(* Logix 5000 project; controller WWTP_SEC_CLX vendor 1 type 14 code 54 rev 17.2; software revision 17.00 *)
// WWTP Secondary Treatment System

TASK MainTask (continuous, watchdog 500 ms) : MainProgram, SecTank01_Drive, SecTank02_Drive, AerationBlower, SecTank01_RAS_Pump

MODULES
   Local : vendor 1 type 14 code 54 (ICP 0, rev 17.2)
      WWTP_SEC_CLX_Rack00_Slot02_DI : 1756-IA16 (ICP 2, rev 3.2, Input RPI 20 ms)
           Local:2:I.DATA.4   // Secondary Tank #1 In-Auto
           Local:2:I.DATA.7   // Secondary Tank #2 In-Auto
           Local:2:I.DATA.0   // BLR-400 In-Auto
           Local:2:I.DATA.1   // BLR-400 Running
           Local:2:I.DATA.14   // M-401 In-Auto
           Local:2:I.DATA.10   // M-400 Fault
           Local:2:I.DATA.11   // M-400 In-Auto
           Local:2:I.DATA.12   // M-401 Running
           Local:2:I.DATA.13   // M-401 Fault
           Local:2:I.DATA.2   // BLR-400 Fault
           Local:2:I.DATA.9   // M-400 Running
           Local:2:I.DATA.5   // Secondary Tank #1 Torque
           Local:2:I.DATA.8   // Secondary Tank #2 Torque
           Local:2:I.DATA.6   // Secondary Tank #2 Running
           Local:2:I.DATA.3   // Secondary Tank #1 Running
      WWTP_SEC_CLS_Rack00_Slot03_DI : 1756-IA16 (ICP 3, rev 3.2, Input RPI 20 ms)
           Local:3:I.DATA.4   // M-403 Fault
           Local:3:I.DATA.5   // M-403 In-Auto
           Local:3:I.DATA.0   // M-402 Running
           Local:3:I.DATA.3   // M-403 Running
           Local:3:I.DATA.1   // M-402 Fault
           Local:3:I.DATA.2   // M-402 In-Auto
      WWTP_SEC_CLX_Rack00_Slot04_DO : vendor 1 type 7 code 13 (ICP 4, rev 3.2, Output RPI 20 ms)
           Local:4:O.DATA.5   // M-402 Start/Stop
           Local:4:O.DATA.1   // Secondary Tank #2 Start/Stop
           Local:4:O.DATA.2   // BLR-400 Start/Stop
           Local:4:O.DATA.3   // M-400 Start/Stop
           Local:4:O.DATA.4   // M-401 Start/Stop
           Local:4:O.DATA.0   // Secondary Tank #1 Start/Stop
           Local:4:O.DATA.6   // M-403 Start/Stop
      WWTP_SEC_CLX_Rack00_Slot05_AI : 1756-IF16 (ICP 5, rev 1.5, Input RPI 100 ms)
           Local:5:I.CH1DATA   // Secondary Tank #2 RAS Control 0 - 3 MGD
           Local:5:I.CH0DATA   // Secondary Tank #1 RAS Control 0 - 3 MGD
      WWTP_SEC_CLX_Rack00_Slot01_ENBT : 1756-ENBT (Ethernet 10.16.3.230, ICP 1, rev 4.2)
         WWTP_RAS_P401 : vendor 1 type 123 code 104 (Ethernet 10.16.3.233, rev 6.4, Output RPI 20 ms)
END_MODULES

TYPE STRING_16 :
STRUCT
   LEN : DINT;
   DATA : SINT[16];
END_STRUCT
END_TYPE

TYPE STRING_20 :
STRUCT
   LEN : DINT;
   DATA : SINT[20];
END_STRUCT
END_TYPE

TYPE STRING_40 :
STRUCT
   LEN : DINT;
   DATA : SINT[40];
END_STRUCT
END_TYPE

TYPE STRING_8 :
STRUCT
   LEN : DINT;
   DATA : SINT[8];
END_STRUCT
END_TYPE

ADD_ON_INSTRUCTION P_AIn   (* revision 0.31, ExecutePrescan, ExecuteEnableInFalse *)
// Analog Input
// Revision note:
// Fixed handling of +/- Inf (1.$) and +/- NaN (1.#QNAN) on Val_InpPV, Val, and filter.
// Help:
// This Instruction monitors an Analog Input from a flow, level, pressure,
// temperature, or any other analog sensor, and provides:
// *  Scaling, from Input (Raw) to PV (Engineering) Units
// *  High-High, High, Low and Low-Low Alarms with configurable delay times and deadbands
// *  Monitoring of input uncertain/bad variable/communication status and out-of-range conditions with alarm
// *  Setting of a simulated input signal for process simulation
// Modes of operation: Operator, Program, Maintenance
// *  Program and Operator Settings for Alarm Thresholds
// *  Maintenance Commands to allow manual override of the input signal (Substitute PV)
VAR_INPUT
   Inp_PV : REAL; {visible}   // Input Signal (process variable) from Sensor
   Inp_PVBad : BOOL;   // 1=PV or I/O Comms Status Bad, 0=OK
   Inp_PVUncertain : BOOL;   // 1=PV Value Not Reliable, 0=OK
   Inp_Sim : BOOL;   // 1=Use simulated PV (Set_SimPV); 0=Use Input (Inp_PV)
   Inp_Reset : BOOL;   // 1=Reset all Alarms requiring reset
   Cfg_NoSubstPV : BOOL;   // 1=Disallow selection of Substitute PV
   Cfg_SetTrack : BOOL := 1;   // 1=PSets track OSets in Oper, OSets track PSets in Prog, 0=no tracking
   Cfg_PCmdClear : BOOL := 1;   // 1=Clear Program Commands on receipt 0=Leave Set
   Cfg_HasHiHiAlm : BOOL;   // 1=High-High Alarm exists and will be checked
   Cfg_HasHiAlm : BOOL;   // 1=High Alarm exists and will be checked
   Cfg_HasLoAlm : BOOL;   // 1=Low Alarm exists and will be checked
   Cfg_HasLoLoAlm : BOOL;   // 1=Low-Low Alarm exists and will be checked
   Cfg_HasFailAlm : BOOL;   // 1=Analog Input Failure Alarm exists and will be checked
   Cfg_HiHiResetReqd : BOOL;   // 1=Reset required to clear High-High Alarm
   Cfg_HiResetReqd : BOOL;   // 1=Reset required to clear High Alarm
   Cfg_LoResetReqd : BOOL;   // 1=Reset required to clear Low Alarm
   Cfg_LoLoResetReqd : BOOL;   // 1=Reset required to clear Low-Low Alarm
   Cfg_FailResetReqd : BOOL;   // 1=Reset required to clear Analog InputFailure Alarm
   Cfg_HiHiAckReqd : BOOL := 1;   // 1=Acknowledge required for High-High Alarm
   Cfg_HiAckReqd : BOOL := 1;   // 1=Acknowledge required for High Alarm
   Cfg_LoAckReqd : BOOL := 1;   // 1=Acknlowledge required for Low Alarm
   Cfg_LoLoAckReqd : BOOL := 1;   // 1=Acknowledge required for Low-Low Alarm
   Cfg_FailAckReqd : BOOL := 1;   // 1=Acknowledge required for Analog Input Failure Alarm
   Cfg_HiHiSeverity : SINT := 3;   // High-High Alarm Severity 1=info, 2=warn, 3=excep, 4=fault
   Cfg_HiSeverity : SINT := 2;   // High Alarm Severity 1=info, 2=warn, 3=excep, 4=fault
   Cfg_LoSeverity : SINT := 2;   // Low Alarm Severity 1=info, 2=warn, 3=excep, 4=fault
   Cfg_LoLoSeverity : SINT := 3;   // Low-Low Alarm Severity 1=info, 2=warn, 3=excep, 4=fault
   Cfg_FailSeverity : SINT := 4;   // Failure Alarm Severity 1=info, 2=warn, 3=excep, 4=fault
   Cfg_InpRawMin : REAL;   // Input (unscaled) Minimum for Scaling
   Cfg_InpRawMax : REAL := 100.0;   // Input (unscaled) Maximum for Scaling
   Cfg_PVEUMin : REAL;   // PV (Output) Minimum for Scaling to EU
   Cfg_PVEUMax : REAL := 100.0;   // PV (Output) Maximum for Scaling to EU
   Cfg_FiltTC : REAL;   // PV Filter Time Constant (sec), 0.0 = unfiltered
   Cfg_HiHiDB : REAL := 1.0;   // High-High Alarm Deadband (EU)
   Cfg_HiHiMinDuration : DINT;   // Minimum time above High-High Limit to raise Alarm (sec)
   Cfg_HiDB : REAL := 1.0;   // High Alarm Deadband (EU)
   Cfg_HiMinDuration : DINT;   // Minimum time above High Limit to raise Alarm (sec)
   Cfg_LoDB : REAL := 1.0;   // Low Alarm Deadband (EU)
   Cfg_LoMinDuration : DINT;   // Minimum time below Low Limit to raise Alarm (sec)
   Cfg_LoLoDB : REAL := 1.0;   // Low-Low Alarm Deadband (EU)
   Cfg_LoLoMinDuration : DINT;   // Minimum time below Low-Low Limit to raise Alarm (sec)
   Cfg_FailHiLim : REAL := 1.5e+38;   // Out-of-Range (fail) High Limit (EU)
   Cfg_FailLoLim : REAL := -1.5e+38;   // Out-of-Range (fail) Low Limit (EU)
   Cfg_FailDB : REAL;   // Out-of-Range (fail) High/Low Deadband (EU)
   Cfg_FailMinDuration : DINT;   // Minimum time Bad or Out of Range to raise Fail Alarm (sec)
   PSet_Owner : DINT;   // Program Owner Request ID (non-zero) or Release (zero)
   PSet_HiHiLim : REAL := 1.5e+38;   // Program-Entered High-High Alarm Threshold (EU)
   PSet_HiLim : REAL := 1.5e+38;   // Program-Entered High Alarm Threshold (EU)
   PSet_LoLim : REAL := -1.5e+38;   // Program-Entered Low Alarm Threshold (EU)
   PSet_LoLoLim : REAL := -1.5e+38;   // Program-Entered Low-Low Alarm Threshold (EU)
   MSet_SubstPV : REAL;   // Maintenance-Entered Substitute PV (EU)
   OSet_HiHiLim : REAL := 1.5e+38;   // Operator-Entered High-High Alarm Threshold (EU)
   OSet_HiLim : REAL := 1.5e+38;   // Operator-Entered High Alarm Threshold (EU)
   OSet_LoLim : REAL := -1.5e+38;   // Operator-Entered Low Alarm Threshold (EU)
   OSet_LoLoLim : REAL := -1.5e+38;   // Operator-Entered Low-Low Alarm Threshold (EU)
   Set_SimPV : REAL;   // PV used in Simulation (Inp_Sim=1) (EU)
   PCmd_Acq : BOOL;   // Program Command to Acquire ownership (Oper to Prog)
   PCmd_Rel : BOOL;   // Program Command to Release ownership (Prog to Oper)
   PCmd_Lock : BOOL;   // Program Command to Lock Mode in Prog
   PCmd_Unlock : BOOL;   // Program Command to Unlock Mode
   PCmd_Reset : BOOL;   // Program Command to Reset all Alarms requiring Reset
   PCmd_HiHiAck : BOOL;   // Program Command to Acknowledge High-High Alarm
   PCmd_HiHiInhibit : BOOL;   // Program Command to Inhibit High-High Alarm
   PCmd_HiHiUninhibit : BOOL;   // Program Command to UninhibitHigh-High Alarm
   PCmd_HiAck : BOOL;   // Program Command to Acknowledge High Alarm
   PCmd_HiInhibit : BOOL;   // Program Command to Inhibit High Alarm
   PCmd_HiUninhibit : BOOL;   // Program Command to Uninhibit High Alarm
   PCmd_LoAck : BOOL;   // Program Command to Acknowledge Low Alarm
   PCmd_LoInhibit : BOOL;   // Program Command to Inhibit Low Alarm
   PCmd_LoUninhibit : BOOL;   // Program Command to Uninhibit Low Alarm
   PCmd_LoLoAck : BOOL;   // Program Command to Acknowledge Low-Low Alarm
   PCmd_LoLoInhibit : BOOL;   // Program Command to Inhibit Low-Low Alarm
   PCmd_LoLoUninhibit : BOOL;   // Program Command to Uninhibit Low-Low Alarm
   PCmd_FailAck : BOOL;   // Program Command to Acknowldege Analog Input Failure Alarm
   PCmd_FailInhibit : BOOL;   // Program Command to Inhibit Analog Input Failure Alarm
   PCmd_FailUninhibit : BOOL;   // Program Command to Uninhibit Analog Input Failure Alarm
   MCmd_SubstPV : BOOL;   // Maintenance Command to use Substitute PV (override input)
   MCmd_InpPV : BOOL;   // Maintenance Command to use Input PV (normal)
   OCmd_Reset : BOOL;   // Operator Command to Reset all Alarms requiring Reset
END_VAR
VAR_OUTPUT
   Val : REAL; {visible}   // Analog Value (after Substitute PV, if used)
   Val_InpPV : REAL; {visible}   // Analog Input Value (actual, before Substitute PV selection)
   Val_PVEUMin : REAL;   // Minimum of scaled range = MIN (Cfg_PVEUMin, Cfg_PVEUMax)
   Val_PVEUMax : REAL := 100.0;   // Maximum of scaled range = MAX (Cfg_PVEUMin, Cfg_PVEUMax)
   Val_Owner : DINT;   // Current Object Owner ID (0=not owned)
   Val_Notify : SINT;   // Current Alarm Level and Acknowledgement (enumeration)
   Val_HiHiLim : REAL := 1.5e+38; {visible}   // Current High-High Alarm Threshold
   Val_HiLim : REAL := 1.5e+38; {visible}   // Current High Alarm Threshold
   Val_LoLim : REAL := -1.5e+38; {visible}   // Current Low Alarm Threshold
   Val_LoLoLim : REAL := -1.5e+38; {visible}   // Current Low-Low Alarm Threshold
   Sts_SubstPV : BOOL;   // 1=Using Substitute PV (Input being overridden)
   Sts_InpPV : BOOL := 1;   // 1=Using Input PV (normal)
   Sts_PVBad : BOOL;   // 1=PV Bad quality or Out of Range
   Sts_PVUncertain : BOOL;   // 1=PV Value is Uncertain (quality)
   Sts_Err : BOOL; {visible}   // 1=Error in Config, see detail Err_ bits for reason
   Err_Raw : BOOL;   // 1=Error in Config: Raw Input Scaling Min = Max
   Err_EU : BOOL;   // 1=Error in Config: Scaled EU Min = Max
   Err_Filt : BOOL;   // 1=Error in Config: PV filter params (RateTime, TC)
   Err_DB : BOOL;   // 1=Error in Config: an Alarm Deadband is < 0.0
   Err_Alarm : BOOL;   // 1=Error in Config: Invalid Alarm Min Duration or Severity
   Sts_Maint : BOOL;   // 1=Mode is Maintenance (supersedes Prog, Oper)
   Sts_Prog : BOOL;   // 1=Mode is Program
   Sts_Oper : BOOL := 1;   // 1=Mode is Operator
   Sts_ProgOperLock : BOOL;   // 1=Program or Operator has requested Mode Lock
   Sts_HiHi : BOOL;   // 1=Analog Input is above High-High limit
   Alm_HiHi : BOOL;   // 1=Analog Input is in High-High Alarm
   Ack_HiHi : BOOL;   // 1=High-High Alarm has been acknowledged
   Sts_HiHiDisabled : BOOL;   // 1=High-High Alarm is Disabled (not saved or sent)
   Sts_HiHiInhibited : BOOL;   // 1=High-High Alarm is Inhibited by logic
   Sts_HiHiSuppressed : BOOL;   // 1=High-High Alarm has been suppressed (logged only)
   Sts_Hi : BOOL;   // 1=Analog Input is above High limit
   Alm_Hi : BOOL;   // 1=Analog Input is in High Alarm
   Ack_Hi : BOOL;   // 1=High Alarm has been acknowledged
   Sts_HiDisabled : BOOL;   // 1=High Alarm is Disabled (not saved or sent)
   Sts_HiInhibited : BOOL;   // 1=High Alarm is Inhibited by logic
   Sts_HiSuppressed : BOOL;   // 1=High Alarm has been suppressed (logged only)
   Sts_Lo : BOOL;   // 1=Analog Input is below Low limit
   Alm_Lo : BOOL;   // 1=Analog Input is in Low Alarm
   Ack_Lo : BOOL;   // 1=Low Alarm has been acknowledged
   Sts_LoDisabled : BOOL;   // 1=Low Alarm is Disabled (not saved or sent)
   Sts_LoInhibited : BOOL;   // 1=Low Alarm is Inhibited by logic
   Sts_LoSuppressed : BOOL;   // 1=Low Alarm has been suppressed (logged only)
   Sts_LoLo : BOOL;   // 1=Analog Input is below Low-Low limit
   Alm_LoLo : BOOL;   // 1=Analog Input is in Low-Low Alarm
   Ack_LoLo : BOOL;   // 1=Low-Low Alarm has been acknowledged
   Sts_LoLoDisabled : BOOL;   // 1=Low-Low Alarm is Disabled (not saved or sent)
   Sts_LoLoInhibited : BOOL;   // 1=Low-Low Alarm is Inhibited by logic
   Sts_LoLoSuppressed : BOOL;   // 1=Low-Low Alarm has been suppressed (logged only)
   Sts_Fail : BOOL;   // 1=Analog Input is Out of Range or PV Bad
   Alm_Fail : BOOL;   // 1=Analog Input Failure Alarm (Bad or Out of Range)
   Ack_Fail : BOOL;   // 1=Analog Input Failure Alarm has been acknowledged
   Sts_FailDisabled : BOOL;   // 1=Analog input Failure Alarm is Disabled (not saved or sent)
   Sts_FailInhibited : BOOL;   // 1=Analog Input Failure Alarm is inhibited by logic
   Sts_FailSuppressed : BOOL;   // 1=Analog Input Failure Alarm has been suppressed (logged only)
   Rdy_SubstPV : BOOL;   // 1=Ready for MCmd_SubstPV
   Rdy_InpPV : BOOL;   // 1=Ready for MCmd_InpPV
   Rdy_Reset : BOOL;   // 1=At least one Alarm requires Reset
END_VAR
VAR
   LoLo : P_Alarm := (Inp := 1, Cfg_AckReqd := 1, Cfg_Severity := 3, Ack := 1, Rdy_Disable := 1);   // Low-Low Alarm
   Lo : P_Alarm := (Inp := 1, Cfg_AckReqd := 1, Cfg_Severity := 3, Ack := 1, Rdy_Disable := 1);   // Low Alarm
   Hi : P_Alarm := (Inp := 1, Cfg_AckReqd := 1, Cfg_Severity := 2, Ack := 1, Rdy_Disable := 1);   // High Alarm
   HiHi : P_Alarm := (Inp := 1, Cfg_AckReqd := 1, Cfg_Severity := 3, Ack := 1, Rdy_Disable := 1);   // High-High Alarm
   Mode : P_Mode := (Cfg_PCmdClear := 1, Cfg_OvrdOverLock := 1, Sts_Oper := 1, Rdy_Rel := 1, Rdy_AcqLock := 1);   // Analog Input Mode Selection
   Cfg_EU : STRING_8 := '%';   // Engineering Units for display on HMI
   Cfg_Tag : STRING_20 := 'P_AIn';   // Tagname for display on HMI
   Cfg_Label : STRING_20 := 'Analog Input';   // Label for graphic symbol displayed on HMI
   Cfg_Desc : STRING_40 := 'Analog Input';   // Description for display on HMI
   Fail : P_Alarm := (Inp := 1, Cfg_AckReqd := 1, Cfg_Severity := 3, Ack := 1, Rdy_Disable := 1);   // Analog Input Failure Alarm (bad quality or out of range)
   Wrk_Notify : SINT;   // Buffer for building Val_Notify
   Wrk_SubstPV : BOOL;   // Internal flag: Using Substitute PV
   Wrk_UnfiltPV : REAL;   // Unfiltered PV, input to 1st order filter
   Wrk_Alpha : REAL;   // Filter multiplier = (1 / (1+TC/dT) )
   Wrk_ScanT : TIMER := (PRE := 2147483647);   // Scan Timer (milliseconds, always runs)
   Wrk_ScanTime : REAL;   // Time since this instance was last scanned
   Wrk_FiltPV : REAL;   // Filtered PV
   Wrk_InpDINT : DINT;   // Input REAL bit pattern as a DINT (check for Inf/NaN)
   Wrk_InpInfNaN : BOOL;   // Input is Infinite or Not a Number
   Wrk_ValidONS : BOOL;   // Selected PV goes from Infinite or Not a Number to VALID
   Wrk_SelPVDINT : DINT;   // Selected PV check for Infinite or Non A Number
   Wrk_SelPVInfNaN : BOOL;   // Selected PV (Input or Substitute) is Infinite or NaN
END_VAR

ROUTINE EnableInFalse   (* ladder *)
// Off-Scan: no Val update or alarm checking.  PV Bad Quality ("stale") is asserted.
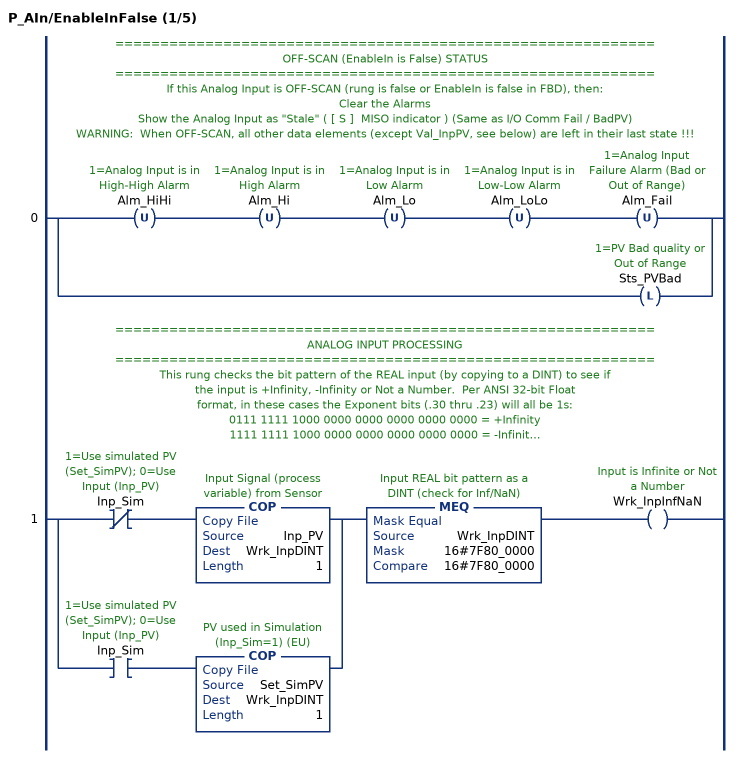
   // ============================================================
   // OFF-SCAN (EnableIn is False) STATUS
   // ============================================================
   // If this Analog Input is OFF-SCAN (rung is false or EnableIn is false in FBD), then:
   // Clear the Alarms
   // Show the Analog Input as "Stale" ( [ S ]  MISO indicator ) (Same as I/O Comm Fail / BadPV)
   // WARNING:  When OFF-SCAN, all other data elements (except Val_InpPV, see below) are left in their last state !!!
   0: [OTU(Alm_HiHi) OTU(Alm_Hi) OTU(Alm_Lo) OTU(Alm_LoLo) OTU(Alm_Fail) ,OTL(Sts_PVBad) ];
   // ============================================================
   // ANALOG INPUT PROCESSING
   // ============================================================
   // This rung checks the bit pattern of the REAL input (by copying to a DINT) to see if
   // the input is +Infinity, -Infinity or Not a Number.  Per ANSI 32-bit Float
   // format, in these cases the Exponent bits (.30 thru .23) will all be 1s:
   // 0111 1111 1000 0000 0000 0000 0000 0000 = +Infinity
   // 1111 1111 1000 0000 0000 0000 0000 0000 = -Infinity
   // x111 1111 1xxx xxxx xxxx xxxx xxxx xxxx = Not a Number
   1: [XIO(Inp_Sim) COP(Inp_PV,Wrk_InpDINT,1) ,XIC(Inp_Sim) COP(Set_SimPV,Wrk_InpDINT,1) ]MEQ(Wrk_InpDINT,16#7F80_0000,16#7F80_0000)OTE(Wrk_InpInfNaN);
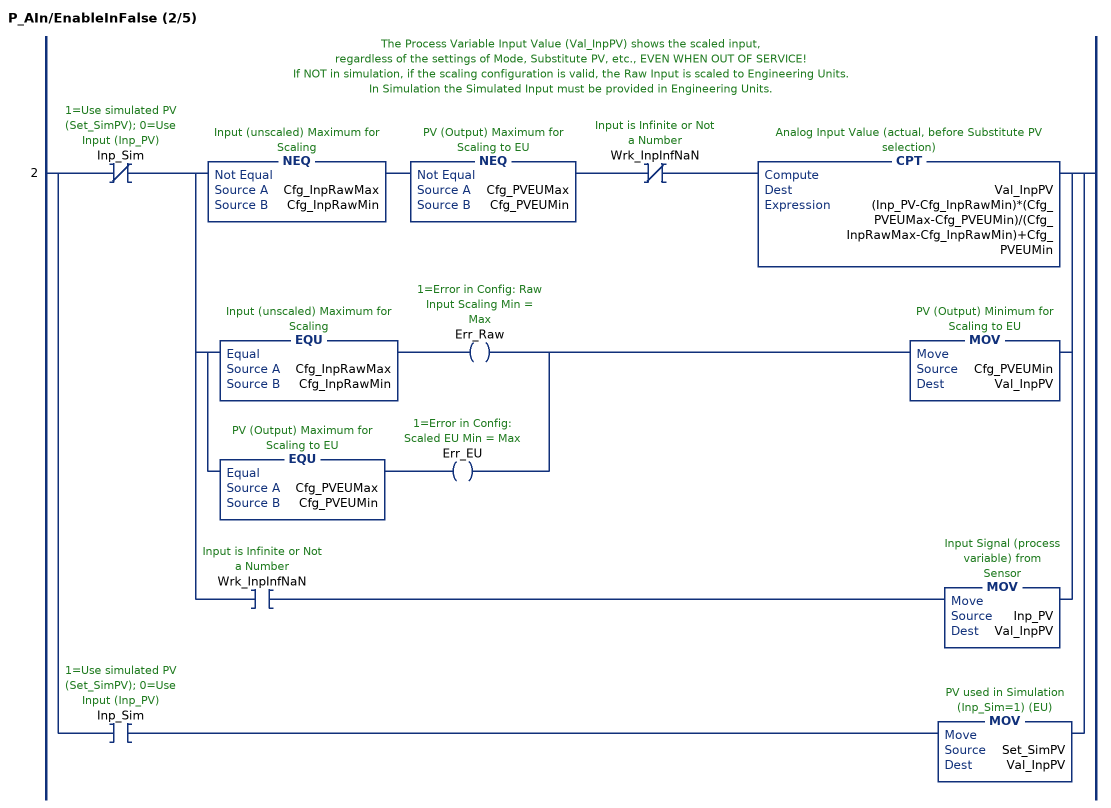
   // The Process Variable Input Value (Val_InpPV) shows the scaled input,
   // regardless of the settings of Mode, Substitute PV, etc., EVEN WHEN OUT OF SERVICE!
   // If NOT in simulation, if the scaling configuration is valid, the Raw Input is scaled to Engineering Units.
   // In Simulation the Simulated Input must be provided in Engineering Units.
   2: [XIO(Inp_Sim) [NEQ(Cfg_InpRawMax,Cfg_InpRawMin) NEQ(Cfg_PVEUMax,Cfg_PVEUMin) XIO(Wrk_InpInfNaN) CPT(Val_InpPV,(Inp_PV-Cfg_InpRawMin)*(Cfg_PVEUMax-Cfg_PVEUMin)/(Cfg_InpRawMax-Cfg_InpRawMin)+Cfg_PVEUMin) ,[EQU(Cfg_InpRawMax,Cfg_InpRawMin) OTE(Err_Raw) ,EQU(Cfg_PVEUMax,Cfg_PVEUMin) OTE(Err_EU) ] MOV(Cfg_PVEUMin,Val_InpPV) ,XIC(Wrk_InpInfNaN) MOV(Inp_PV,Val_InpPV) ] ,XIC(Inp_Sim) MOV(Set_SimPV,Val_InpPV) ];
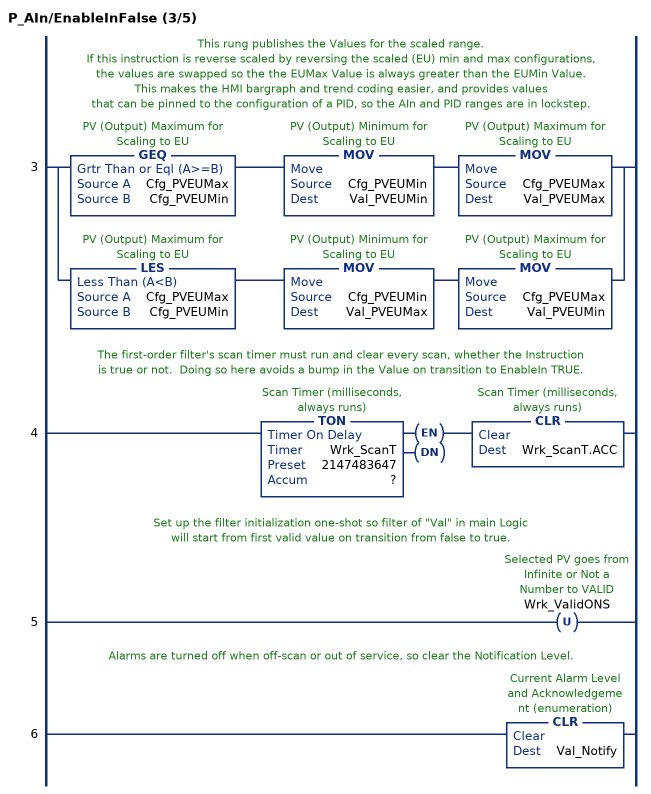
   // This rung publishes the Values for the scaled range.
   // If this instruction is reverse scaled by reversing the scaled (EU) min and max configurations,
   // the values are swapped so the the EUMax Value is always greater than the EUMin Value.
   // This makes the HMI bargraph and trend coding easier, and provides values
   // that can be pinned to the configuration of a PID, so the AIn and PID ranges are in lockstep.
   3: [GEQ(Cfg_PVEUMax,Cfg_PVEUMin) MOV(Cfg_PVEUMin,Val_PVEUMin) MOV(Cfg_PVEUMax,Val_PVEUMax) ,LES(Cfg_PVEUMax,Cfg_PVEUMin) MOV(Cfg_PVEUMin,Val_PVEUMax) MOV(Cfg_PVEUMax,Val_PVEUMin) ];
   // The first-order filter's scan timer must run and clear every scan, whether the Instruction
   // is true or not.  Doing so here avoids a bump in the Value on transition to EnableIn TRUE.
   4: TON(Wrk_ScanT,?,?)CLR(Wrk_ScanT.ACC);
   // Set up the filter initialization one-shot so filter of "Val" in main Logic
   // will start from first valid value on transition from false to true.
   5: OTU(Wrk_ValidONS);
   // Alarms are turned off when off-scan or out of service, so clear the Notification Level.
   6: CLR(Val_Notify);
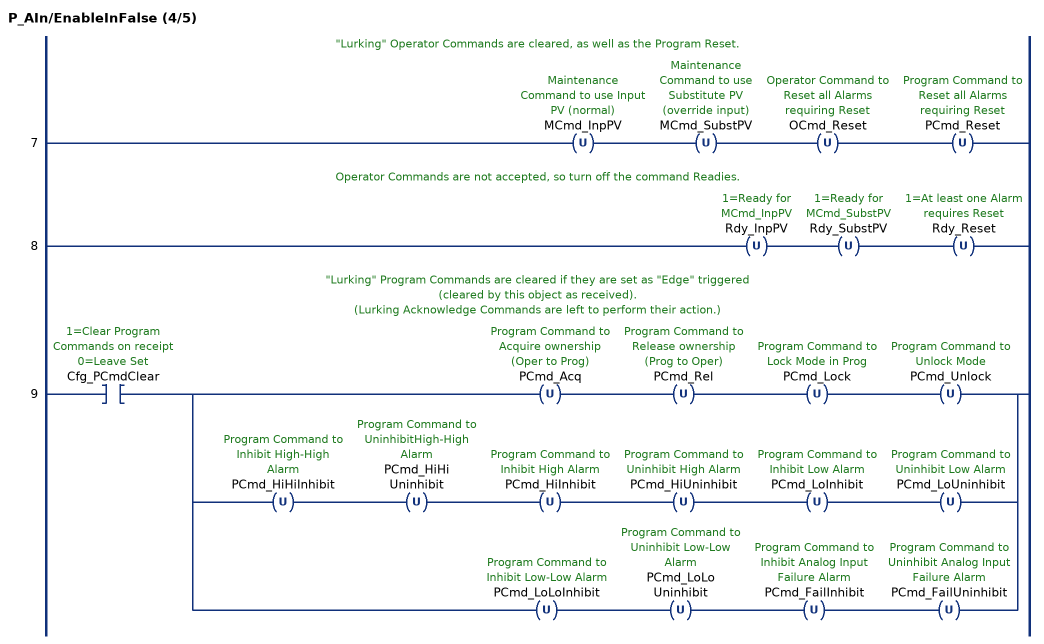
   // "Lurking" Operator Commands are cleared, as well as the Program Reset.
   7: OTU(MCmd_InpPV)OTU(MCmd_SubstPV)OTU(OCmd_Reset)OTU(PCmd_Reset);
   // Operator Commands are not accepted, so turn off the command Readies.
   8: OTU(Rdy_InpPV)OTU(Rdy_SubstPV)OTU(Rdy_Reset);
   // "Lurking" Program Commands are cleared if they are set as "Edge" triggered
   // (cleared by this object as received).
   // (Lurking Acknowledge Commands are left to perform their action.)
   9: XIC(Cfg_PCmdClear)[OTU(PCmd_Acq) OTU(PCmd_Rel) OTU(PCmd_Lock) OTU(PCmd_Unlock) ,OTU(PCmd_HiHiInhibit) OTU(PCmd_HiHiUninhibit) OTU(PCmd_HiInhibit) OTU(PCmd_HiUninhibit) OTU(PCmd_LoInhibit) OTU(PCmd_LoUninhibit) ,OTU(PCmd_LoLoInhibit) OTU(PCmd_LoLoUninhibit) OTU(PCmd_FailInhibit) OTU(PCmd_FailUninhibit) ];
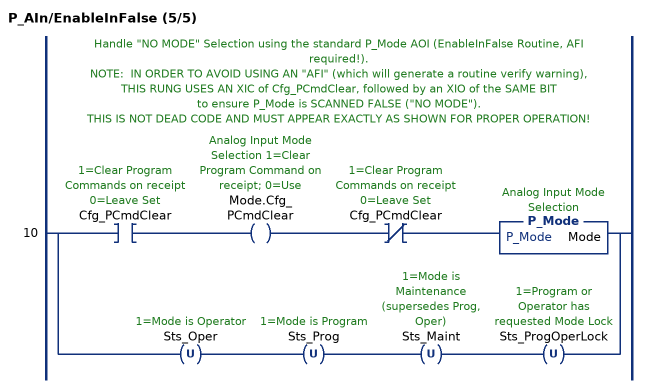
   // Handle "NO MODE" Selection using the standard P_Mode AOI (EnableInFalse Routine, AFI required!).
   // NOTE:  IN ORDER TO AVOID USING AN "AFI" (which will generate a routine verify warning),
   // THIS RUNG USES AN XIC of Cfg_PCmdClear, followed by an XIO of the SAME BIT
   // to ensure P_Mode is SCANNED FALSE ("NO MODE").
   // THIS IS NOT DEAD CODE AND MUST APPEAR EXACTLY AS SHOWN FOR PROPER OPERATION!
   10: [XIC(Cfg_PCmdClear) OTE(Mode.Cfg_PCmdClear) XIO(Cfg_PCmdClear) P_Mode(Mode) ,OTU(Sts_Oper) OTU(Sts_Prog) OTU(Sts_Maint) OTU(Sts_ProgOperLock) ];
END_ROUTINE

ROUTINE Logic   (* ladder *)
// Normal Scan - PV is scaled and alarms are generated
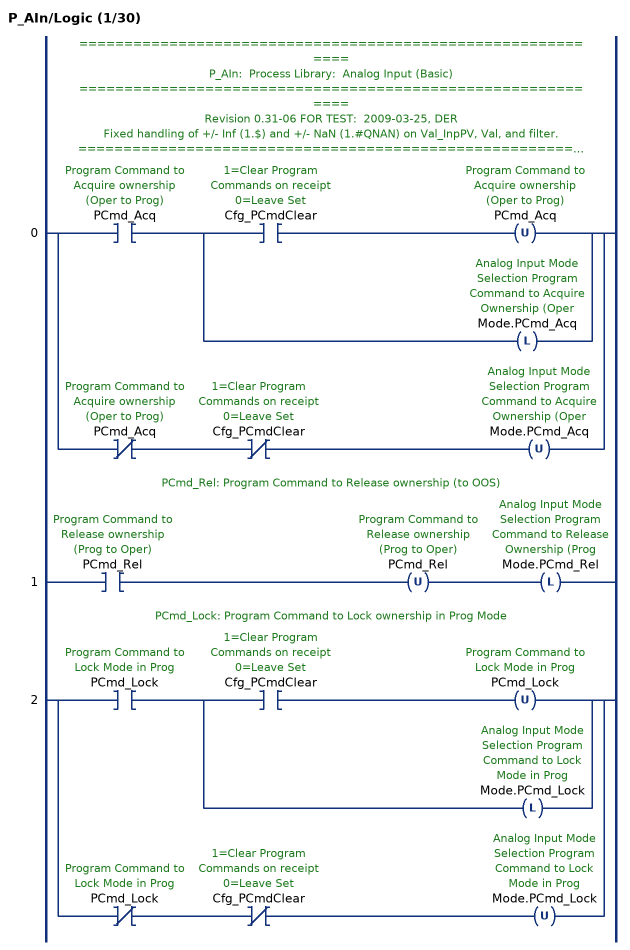
   // ============================================================
   // P_AIn:  Process Library:  Analog Input (Basic)
   // ============================================================
   // Revision 0.31-06 FOR TEST:  2009-03-25, DER
   // Fixed handling of +/- Inf (1.$) and +/- NaN (1.#QNAN) on Val_InpPV, Val, and filter.
   // ============================================================
   // This Instruction monitors an Analog Input from a flow, level, pressure,
   // temperature, or any other analog sensor, and provides:
   // *  Scaling, from Input (Raw) to PV (Engineering) Units
   // *  High-High, High, Low and Low-Low Alarms with configurable delay times and deadbands
   // *  Monitoring of input bad/uncertain variable/communication status and out-of-range conditions with alarm
   // *  Setting of a simulated input signal for process simulation
   // Modes of operation: Operator, Program, Maintenance
   // *  Program and Operator Settings for Alarm Thresholds
   // *  Maintenance Commands to allow manual override of the input signal (Substitute PV)
   // ============================================================
   // POWERUP / INVALID STATE HANDLING
   // ============================================================
   // See Prescan routine for powerup code required for this object.
   // ============================================================
   // MODE PROCESSING
   // ============================================================
   // These rungs handle received Mode Inputs and Commands:
   // NOTE:  Operator Commands for Mode, Alarm are sent directly to the contained P_Mode and P_Alarm AOIs.
   // PCmd_Acq: Program Command to Acquire ownership
   0: [XIC(PCmd_Acq) [XIC(Cfg_PCmdClear) OTU(PCmd_Acq) ,OTL(Mode.PCmd_Acq) ] ,XIO(PCmd_Acq) XIO(Cfg_PCmdClear) OTU(Mode.PCmd_Acq) ];
   // PCmd_Rel: Program Command to Release ownership (to OOS)
   1: XIC(PCmd_Rel)OTU(PCmd_Rel)OTL(Mode.PCmd_Rel);
   // PCmd_Lock: Program Command to Lock ownership in Prog Mode
   2: [XIC(PCmd_Lock) [XIC(Cfg_PCmdClear) OTU(PCmd_Lock) ,OTL(Mode.PCmd_Lock) ] ,XIO(PCmd_Lock) XIO(Cfg_PCmdClear) OTU(Mode.PCmd_Lock) ];
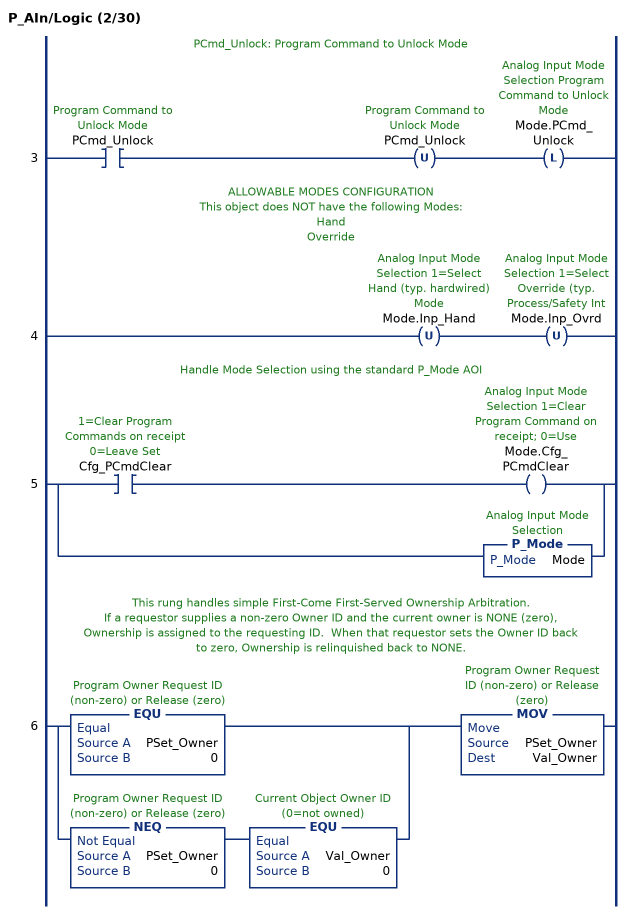
   // PCmd_Unlock: Program Command to Unlock Mode
   3: XIC(PCmd_Unlock)OTU(PCmd_Unlock)OTL(Mode.PCmd_Unlock);
   // ALLOWABLE MODES CONFIGURATION
   // This object does NOT have the following Modes:
   // Hand
   // Override
   4: OTU(Mode.Inp_Hand)OTU(Mode.Inp_Ovrd);
   // Handle Mode Selection using the standard P_Mode AOI
   5: [XIC(Cfg_PCmdClear) OTE(Mode.Cfg_PCmdClear) ,P_Mode(Mode) ];
   // This rung handles simple First-Come First-Served Ownership Arbitration.
   // If a requestor supplies a non-zero Owner ID and the current owner is NONE (zero),
   // Ownership is assigned to the requesting ID.  When that requestor sets the Owner ID back
   // to zero, Ownership is relinquished back to NONE.
   6: [EQU(PSet_Owner,0) ,NEQ(PSet_Owner,0) EQU(Val_Owner,0) ]MOV(PSet_Owner,Val_Owner);
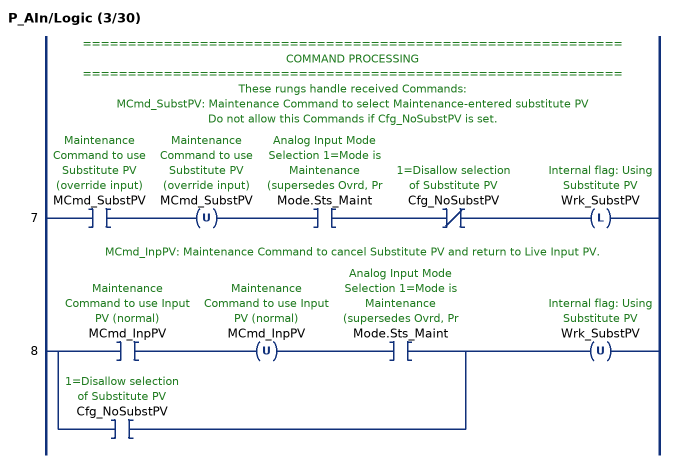
   // ============================================================
   // COMMAND PROCESSING
   // ============================================================
   // These rungs handle received Commands:
   // MCmd_SubstPV: Maintenance Command to select Maintenance-entered substitute PV
   // Do not allow this Commands if Cfg_NoSubstPV is set.
   7: XIC(MCmd_SubstPV)OTU(MCmd_SubstPV)XIC(Mode.Sts_Maint)XIO(Cfg_NoSubstPV)OTL(Wrk_SubstPV);
   // MCmd_InpPV: Maintenance Command to cancel Substitute PV and return to Live Input PV.
   8: [XIC(MCmd_InpPV) OTU(MCmd_InpPV) XIC(Mode.Sts_Maint) ,XIC(Cfg_NoSubstPV) ]OTU(Wrk_SubstPV);
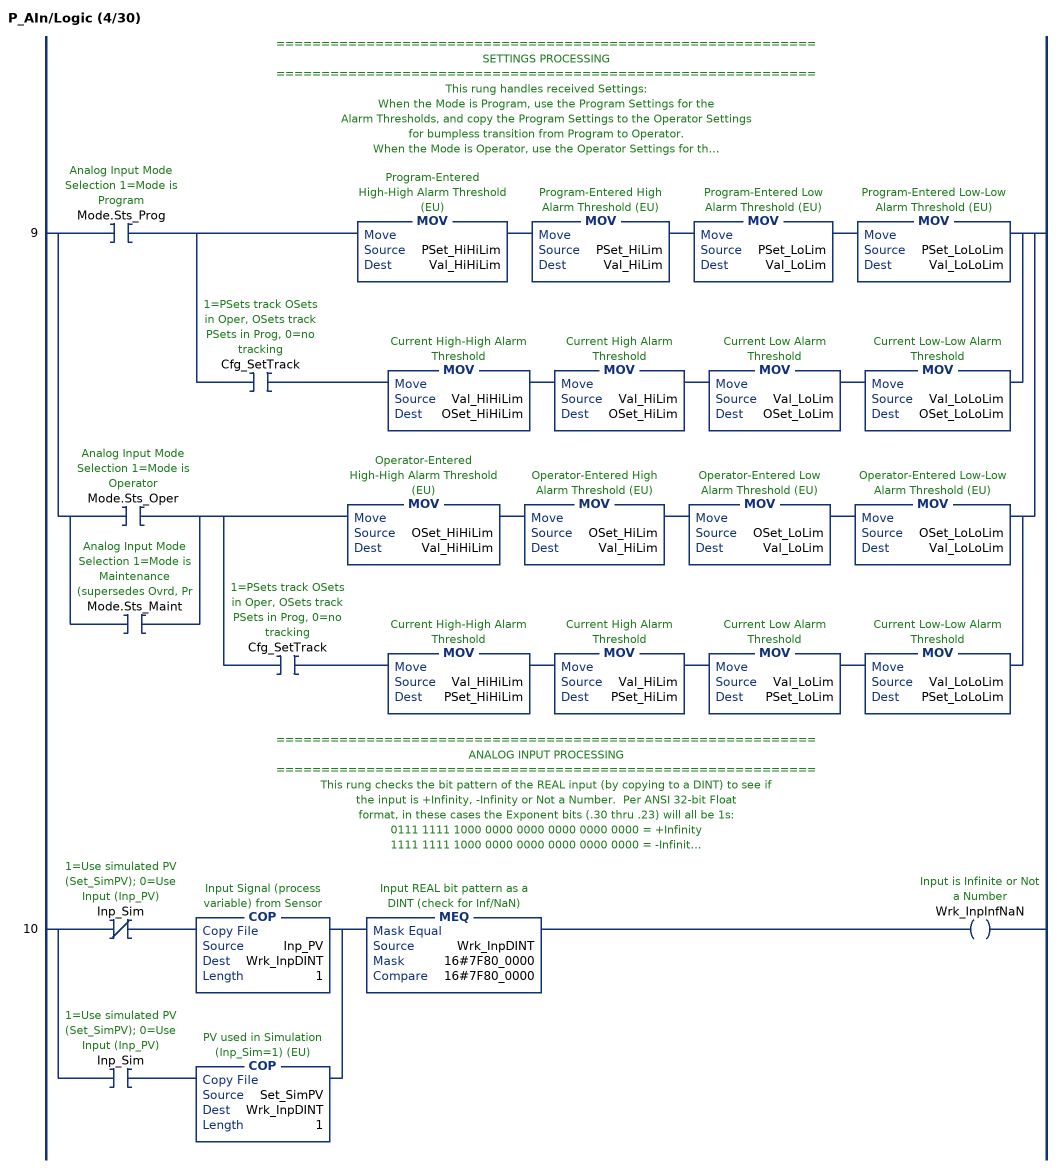
   // ============================================================
   // SETTINGS PROCESSING
   // ============================================================
   // This rung handles received Settings:
   // When the Mode is Program, use the Program Settings for the
   // Alarm Thresholds, and copy the Program Settings to the Operator Settings
   // for bumpless transition from Program to Operator.
   // When the Mode is Operator, use the Operator Settings for the
   // Alarm Thresholds, and copy the Operator Settings to the Program Settings
   // for bumpless transition from Operator to Program.
   9: [XIC(Mode.Sts_Prog) [MOV(PSet_HiHiLim,Val_HiHiLim) MOV(PSet_HiLim,Val_HiLim) MOV(PSet_LoLim,Val_LoLim) MOV(PSet_LoLoLim,Val_LoLoLim) ,XIC(Cfg_SetTrack) MOV(Val_HiHiLim,OSet_HiHiLim) MOV(Val_HiLim,OSet_HiLim) MOV(Val_LoLim,OSet_LoLim) MOV(Val_LoLoLim,OSet_LoLoLim) ] ,[XIC(Mode.Sts_Oper) ,XIC(Mode.Sts_Maint) ] [MOV(OSet_HiHiLim,Val_HiHiLim) MOV(OSet_HiLim,Val_HiLim) MOV(OSet_LoLim,Val_LoLim) MOV(OSet_LoLoLim,Val_LoLoLim) ,XIC(Cfg_SetTrack) MOV(Val_HiHiLim,PSet_HiHiLim) MOV(Val_HiLim,PSet_HiLim) MOV(Val_LoLim,PSet_LoLim) MOV(Val_LoLoLim,PSet_LoLoLim) ] ];
   // ============================================================
   // ANALOG INPUT PROCESSING
   // ============================================================
   // This rung checks the bit pattern of the REAL input (by copying to a DINT) to see if
   // the input is +Infinity, -Infinity or Not a Number.  Per ANSI 32-bit Float
   // format, in these cases the Exponent bits (.30 thru .23) will all be 1s:
   // 0111 1111 1000 0000 0000 0000 0000 0000 = +Infinity
   // 1111 1111 1000 0000 0000 0000 0000 0000 = -Infinity
   // x111 1111 1xxx xxxx xxxx xxxx xxxx xxxx = Not a Number
   10: [XIO(Inp_Sim) COP(Inp_PV,Wrk_InpDINT,1) ,XIC(Inp_Sim) COP(Set_SimPV,Wrk_InpDINT,1) ]MEQ(Wrk_InpDINT,16#7F80_0000,16#7F80_0000)OTE(Wrk_InpInfNaN);
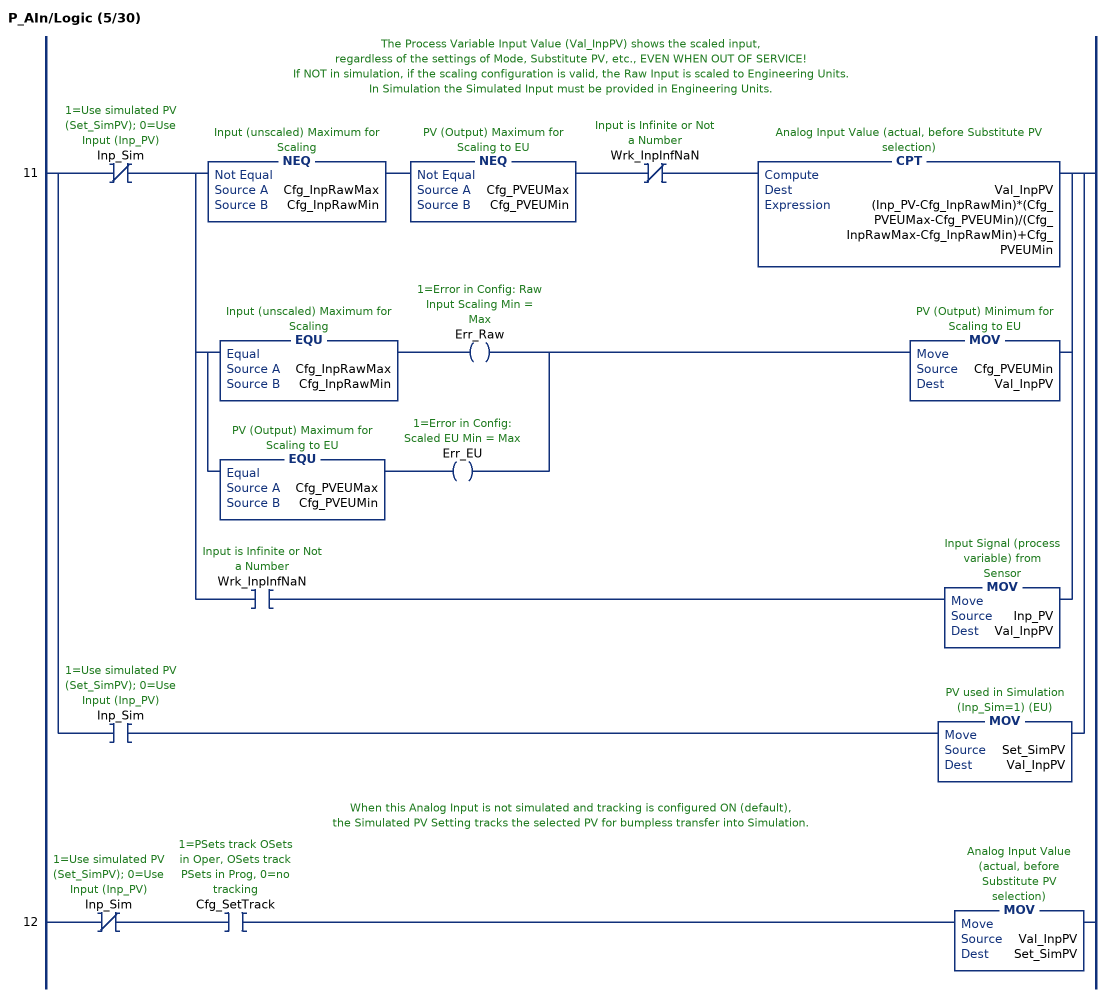
   // The Process Variable Input Value (Val_InpPV) shows the scaled input,
   // regardless of the settings of Mode, Substitute PV, etc., EVEN WHEN OUT OF SERVICE!
   // If NOT in simulation, if the scaling configuration is valid, the Raw Input is scaled to Engineering Units.
   // In Simulation the Simulated Input must be provided in Engineering Units.
   11: [XIO(Inp_Sim) [NEQ(Cfg_InpRawMax,Cfg_InpRawMin) NEQ(Cfg_PVEUMax,Cfg_PVEUMin) XIO(Wrk_InpInfNaN) CPT(Val_InpPV,(Inp_PV-Cfg_InpRawMin)*(Cfg_PVEUMax-Cfg_PVEUMin)/(Cfg_InpRawMax-Cfg_InpRawMin)+Cfg_PVEUMin) ,[EQU(Cfg_InpRawMax,Cfg_InpRawMin) OTE(Err_Raw) ,EQU(Cfg_PVEUMax,Cfg_PVEUMin) OTE(Err_EU) ] MOV(Cfg_PVEUMin,Val_InpPV) ,XIC(Wrk_InpInfNaN) MOV(Inp_PV,Val_InpPV) ] ,XIC(Inp_Sim) MOV(Set_SimPV,Val_InpPV) ];
   // When this Analog Input is not simulated and tracking is configured ON (default),
   // the Simulated PV Setting tracks the selected PV for bumpless transfer into Simulation.
   12: XIO(Inp_Sim)XIC(Cfg_SetTrack)MOV(Val_InpPV,Set_SimPV);
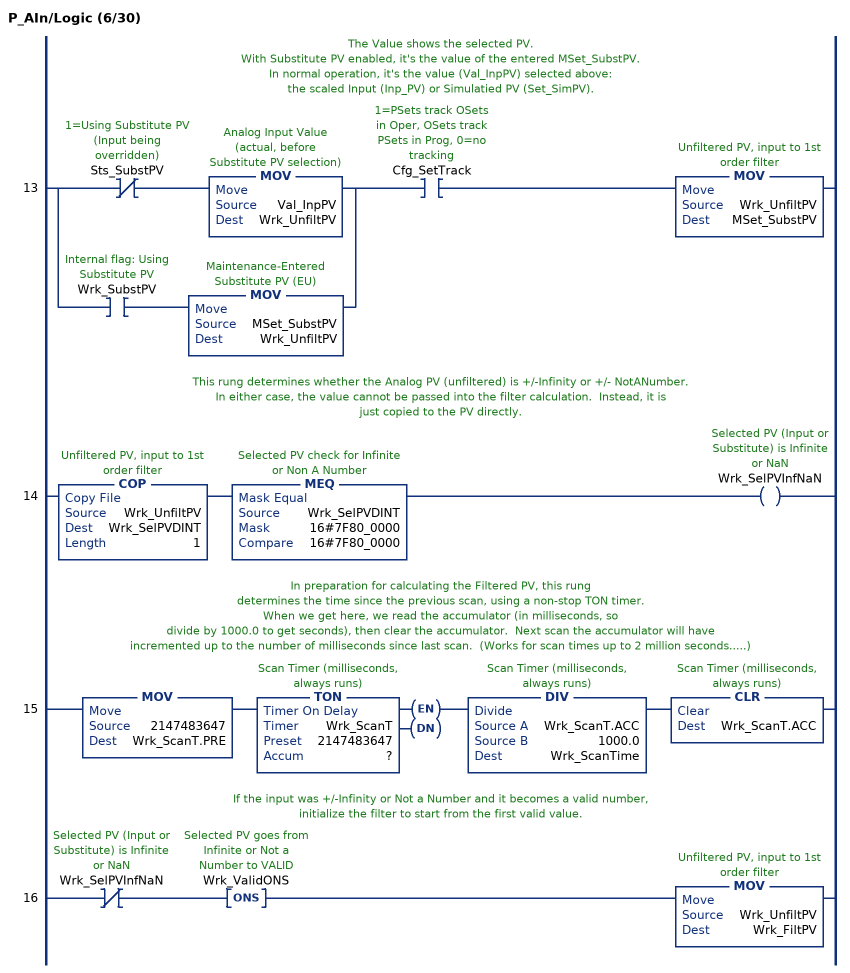
   // The Value shows the selected PV.
   // With Substitute PV enabled, it's the value of the entered MSet_SubstPV.
   // In normal operation, it's the value (Val_InpPV) selected above:
   // the scaled Input (Inp_PV) or Simulatied PV (Set_SimPV).
   13: [XIO(Sts_SubstPV) MOV(Val_InpPV,Wrk_UnfiltPV) ,XIC(Wrk_SubstPV) MOV(MSet_SubstPV,Wrk_UnfiltPV) ]XIC(Cfg_SetTrack)MOV(Wrk_UnfiltPV,MSet_SubstPV);
   // This rung determines whether the Analog PV (unfiltered) is +/-Infinity or +/- NotANumber.
   // In either case, the value cannot be passed into the filter calculation.  Instead, it is
   // just copied to the PV directly.
   14: COP(Wrk_UnfiltPV,Wrk_SelPVDINT,1)MEQ(Wrk_SelPVDINT,16#7F80_0000,16#7F80_0000)OTE(Wrk_SelPVInfNaN);
   // In preparation for calculating the Filtered PV, this rung
   // determines the time since the previous scan, using a non-stop TON timer.
   // When we get here, we read the accumulator (in milliseconds, so
   // divide by 1000.0 to get seconds), then clear the accumulator.  Next scan the accumulator will have
   // incremented up to the number of milliseconds since last scan.  (Works for scan times up to 2 million seconds.....)
   15: MOV(2147483647,Wrk_ScanT.PRE)TON(Wrk_ScanT,?,?)DIV(Wrk_ScanT.ACC,1000.0,Wrk_ScanTime)CLR(Wrk_ScanT.ACC);
   // If the input was +/-Infinity or Not a Number and it becomes a valid number,
   // initialize the filter to start from the first valid value.
   16: XIO(Wrk_SelPVInfNaN)ONS(Wrk_ValidONS)MOV(Wrk_UnfiltPV,Wrk_FiltPV);
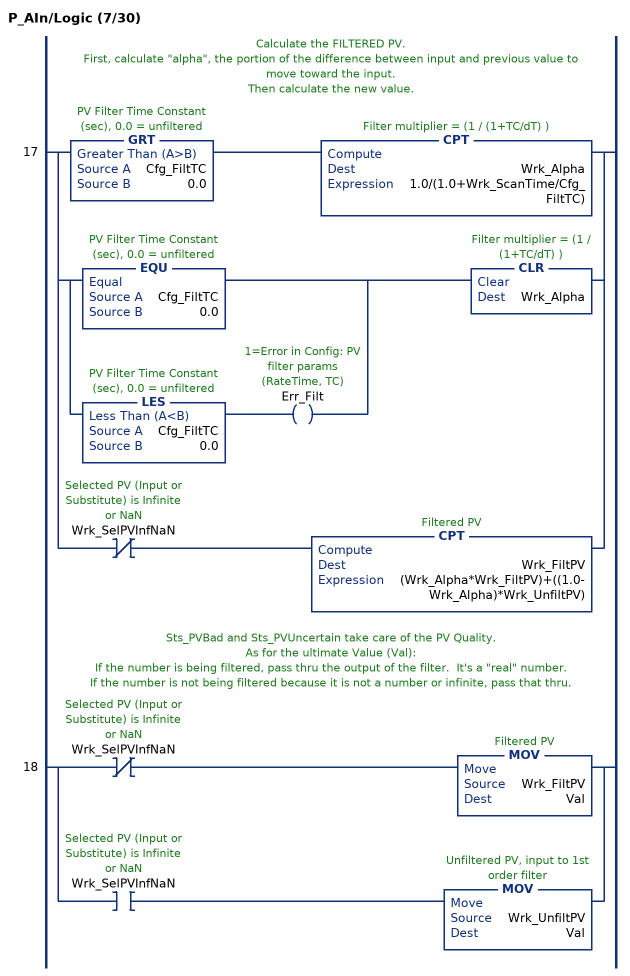
   // Calculate the FILTERED PV.
   // First, calculate "alpha", the portion of the difference between input and previous value to move toward the input.
   // Then calculate the new value.
   17: [GRT(Cfg_FiltTC,0.0) CPT(Wrk_Alpha,1.0/(1.0+Wrk_ScanTime/Cfg_FiltTC)) ,[EQU(Cfg_FiltTC,0.0) ,LES(Cfg_FiltTC,0.0) OTE(Err_Filt) ] CLR(Wrk_Alpha) ,XIO(Wrk_SelPVInfNaN) CPT(Wrk_FiltPV,(Wrk_Alpha*Wrk_FiltPV)+((1.0-Wrk_Alpha)*Wrk_UnfiltPV)) ];
   // Sts_PVBad and Sts_PVUncertain take care of the PV Quality.
   // As for the ultimate Value (Val):
   // If the number is being filtered, pass thru the output of the filter.  It's a "real" number.
   // If the number is not being filtered because it is not a number or infinite, pass that thru.
   18: [XIO(Wrk_SelPVInfNaN) MOV(Wrk_FiltPV,Val) ,XIC(Wrk_SelPVInfNaN) MOV(Wrk_UnfiltPV,Val) ];
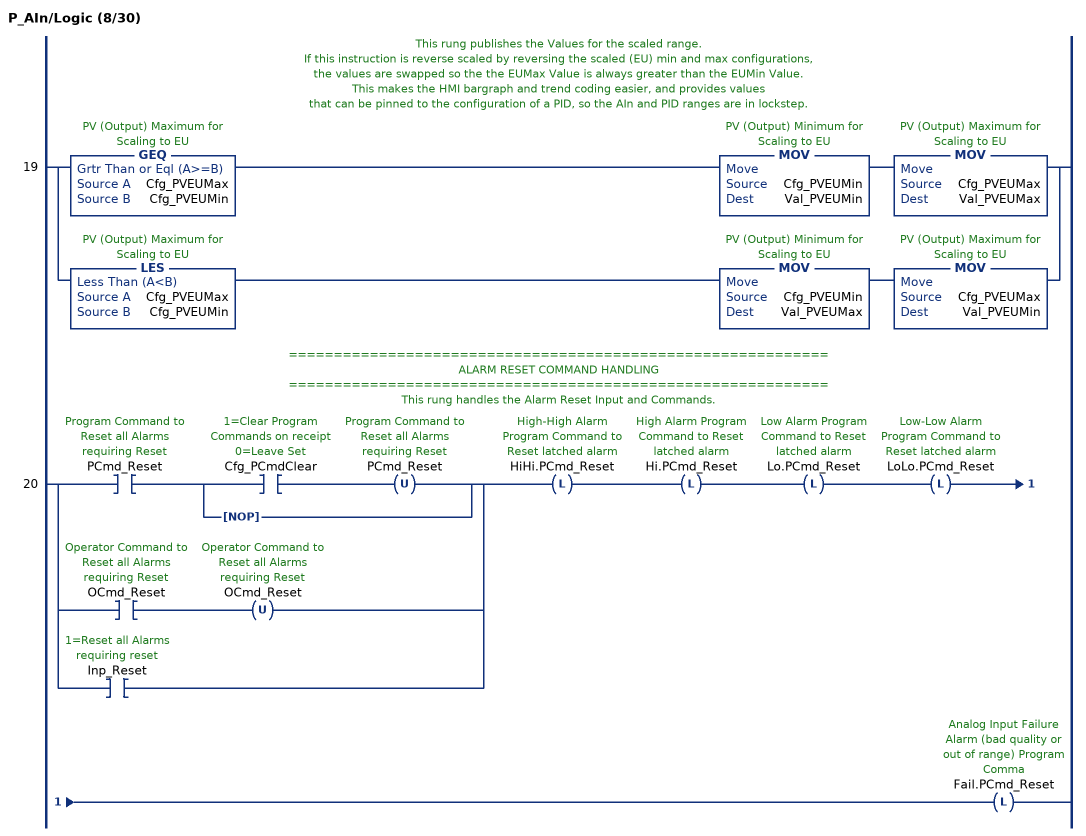
   // This rung publishes the Values for the scaled range.
   // If this instruction is reverse scaled by reversing the scaled (EU) min and max configurations,
   // the values are swapped so the the EUMax Value is always greater than the EUMin Value.
   // This makes the HMI bargraph and trend coding easier, and provides values
   // that can be pinned to the configuration of a PID, so the AIn and PID ranges are in lockstep.
   19: [GEQ(Cfg_PVEUMax,Cfg_PVEUMin) MOV(Cfg_PVEUMin,Val_PVEUMin) MOV(Cfg_PVEUMax,Val_PVEUMax) ,LES(Cfg_PVEUMax,Cfg_PVEUMin) MOV(Cfg_PVEUMin,Val_PVEUMax) MOV(Cfg_PVEUMax,Val_PVEUMin) ];
   // ============================================================
   // ALARM RESET COMMAND HANDLING
   // ============================================================
   // This rung handles the Alarm Reset Input and Commands.
   20: [XIC(PCmd_Reset) [XIC(Cfg_PCmdClear) OTU(PCmd_Reset) ,NOP() ] ,XIC(OCmd_Reset) OTU(OCmd_Reset) ,XIC(Inp_Reset) ]OTL(HiHi.PCmd_Reset)OTL(Hi.PCmd_Reset)OTL(Lo.PCmd_Reset)OTL(LoLo.PCmd_Reset)OTL(Fail.PCmd_Reset);
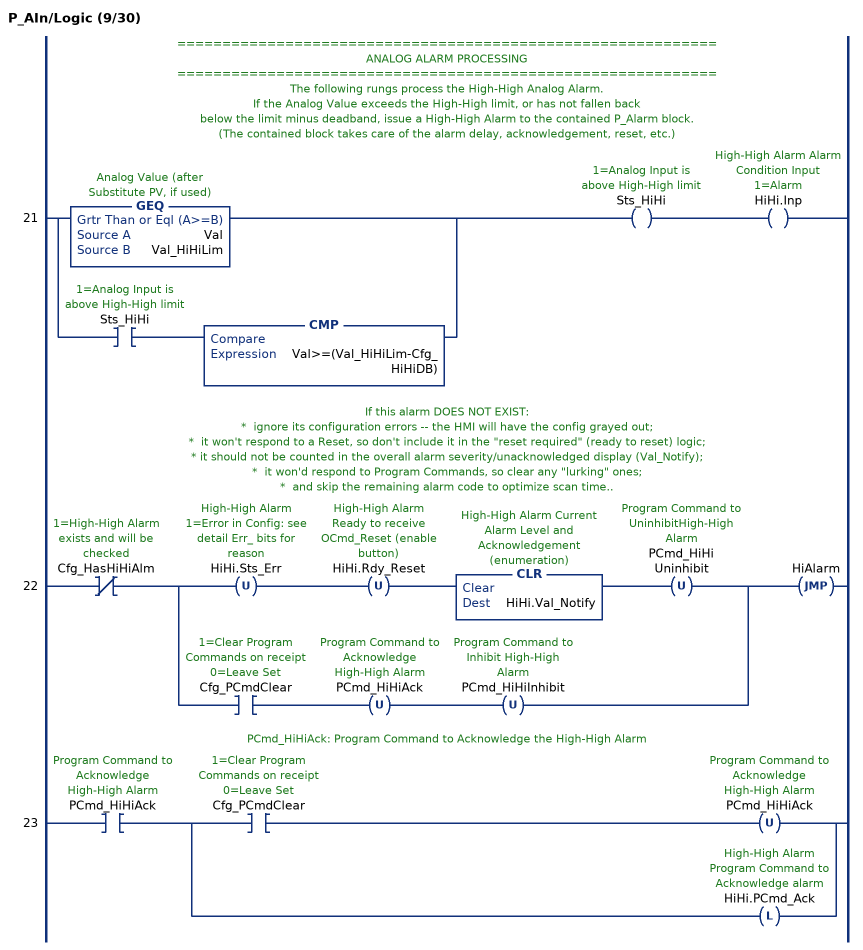
   // ============================================================
   // ANALOG ALARM PROCESSING
   // ============================================================
   // The following rungs process the High-High Analog Alarm.
   // If the Analog Value exceeds the High-High limit, or has not fallen back
   // below the limit minus deadband, issue a High-High Alarm to the contained P_Alarm block.
   // (The contained block takes care of the alarm delay, acknowledgement, reset, etc.)
   21: [GEQ(Val,Val_HiHiLim) ,XIC(Sts_HiHi) CMP(Val>=(Val_HiHiLim-Cfg_HiHiDB)) ]OTE(Sts_HiHi)OTE(HiHi.Inp);
   // If this alarm DOES NOT EXIST:
   // *  ignore its configuration errors -- the HMI will have the config grayed out;
   // *  it won't respond to a Reset, so don't include it in the "reset required" (ready to reset) logic;
   // * it should not be counted in the overall alarm severity/unacknowledged display (Val_Notify);
   // *  it won'd respond to Program Commands, so clear any "lurking" ones;
   // *  and skip the remaining alarm code to optimize scan time..
   22: XIO(Cfg_HasHiHiAlm)[OTU(HiHi.Sts_Err) OTU(HiHi.Rdy_Reset) CLR(HiHi.Val_Notify) OTU(PCmd_HiHiUninhibit) ,XIC(Cfg_PCmdClear) OTU(PCmd_HiHiAck) OTU(PCmd_HiHiInhibit) ]JMP(HiAlarm);
   // PCmd_HiHiAck: Program Command to Acknowledge the High-High Alarm
   23: XIC(PCmd_HiHiAck)[XIC(Cfg_PCmdClear) OTU(PCmd_HiHiAck) ,OTL(HiHi.PCmd_Ack) ];
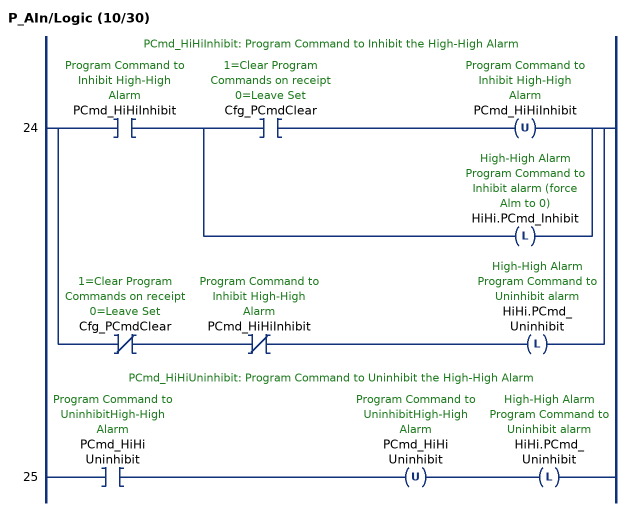
   // PCmd_HiHiInhibit: Program Command to Inhibit the High-High Alarm
   24: [XIC(PCmd_HiHiInhibit) [XIC(Cfg_PCmdClear) OTU(PCmd_HiHiInhibit) ,OTL(HiHi.PCmd_Inhibit) ] ,XIO(Cfg_PCmdClear) XIO(PCmd_HiHiInhibit) OTL(HiHi.PCmd_Uninhibit) ];
   // PCmd_HiHiUninhibit: Program Command to Uninhibit the High-High Alarm
   25: XIC(PCmd_HiHiUninhibit)OTU(PCmd_HiHiUninhibit)OTL(HiHi.PCmd_Uninhibit);
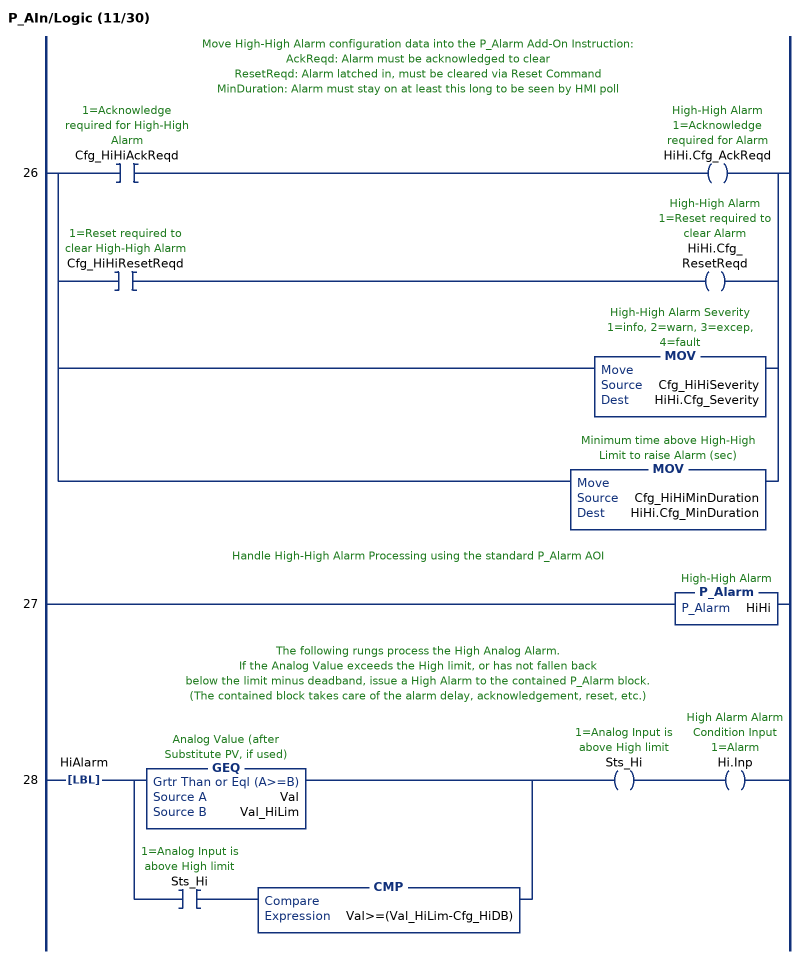
   // Move High-High Alarm configuration data into the P_Alarm Add-On Instruction:
   // AckReqd: Alarm must be acknowledged to clear
   // ResetReqd: Alarm latched in, must be cleared via Reset Command
   // MinDuration: Alarm must stay on at least this long to be seen by HMI poll
   26: [XIC(Cfg_HiHiAckReqd) OTE(HiHi.Cfg_AckReqd) ,XIC(Cfg_HiHiResetReqd) OTE(HiHi.Cfg_ResetReqd) ,MOV(Cfg_HiHiSeverity,HiHi.Cfg_Severity) ,MOV(Cfg_HiHiMinDuration,HiHi.Cfg_MinDuration) ];
   // Handle High-High Alarm Processing using the standard P_Alarm AOI
   27: P_Alarm(HiHi);
   // The following rungs process the High Analog Alarm.
   // If the Analog Value exceeds the High limit, or has not fallen back
   // below the limit minus deadband, issue a High Alarm to the contained P_Alarm block.
   // (The contained block takes care of the alarm delay, acknowledgement, reset, etc.)
   28: LBL(HiAlarm)[GEQ(Val,Val_HiLim) ,XIC(Sts_Hi) CMP(Val>=(Val_HiLim-Cfg_HiDB)) ]OTE(Sts_Hi)OTE(Hi.Inp);
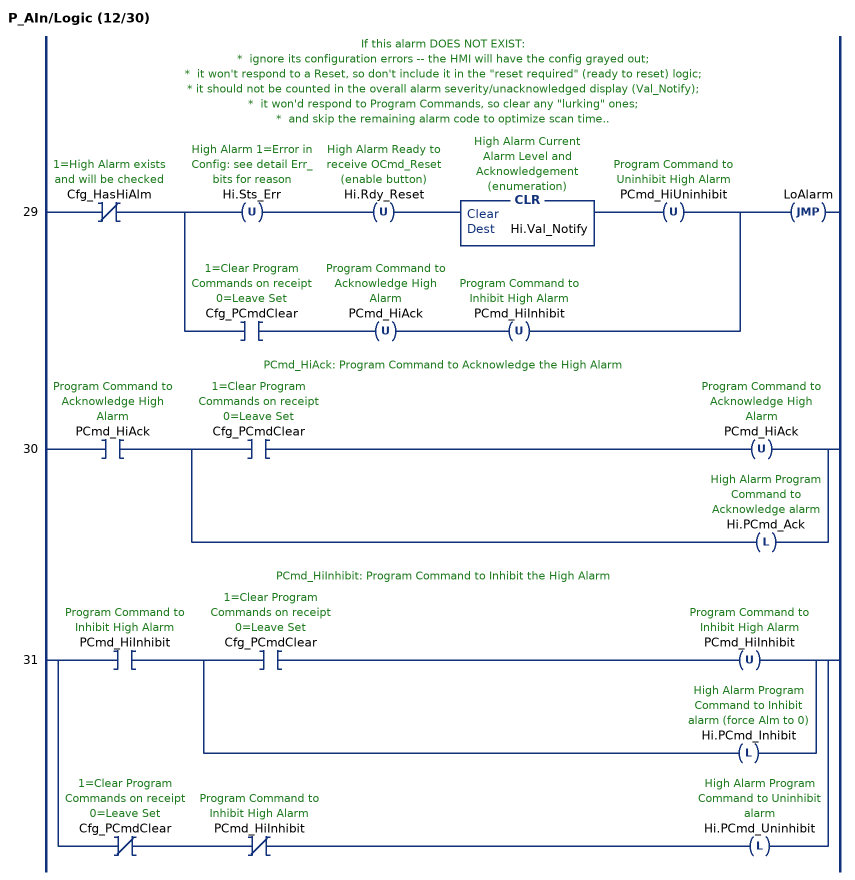
   // If this alarm DOES NOT EXIST:
   // *  ignore its configuration errors -- the HMI will have the config grayed out;
   // *  it won't respond to a Reset, so don't include it in the "reset required" (ready to reset) logic;
   // * it should not be counted in the overall alarm severity/unacknowledged display (Val_Notify);
   // *  it won'd respond to Program Commands, so clear any "lurking" ones;
   // *  and skip the remaining alarm code to optimize scan time..
   29: XIO(Cfg_HasHiAlm)[OTU(Hi.Sts_Err) OTU(Hi.Rdy_Reset) CLR(Hi.Val_Notify) OTU(PCmd_HiUninhibit) ,XIC(Cfg_PCmdClear) OTU(PCmd_HiAck) OTU(PCmd_HiInhibit) ]JMP(LoAlarm);
   // PCmd_HiAck: Program Command to Acknowledge the High Alarm
   30: XIC(PCmd_HiAck)[XIC(Cfg_PCmdClear) OTU(PCmd_HiAck) ,OTL(Hi.PCmd_Ack) ];
   // PCmd_HiInhibit: Program Command to Inhibit the High Alarm
   31: [XIC(PCmd_HiInhibit) [XIC(Cfg_PCmdClear) OTU(PCmd_HiInhibit) ,OTL(Hi.PCmd_Inhibit) ] ,XIO(Cfg_PCmdClear) XIO(PCmd_HiInhibit) OTL(Hi.PCmd_Uninhibit) ];
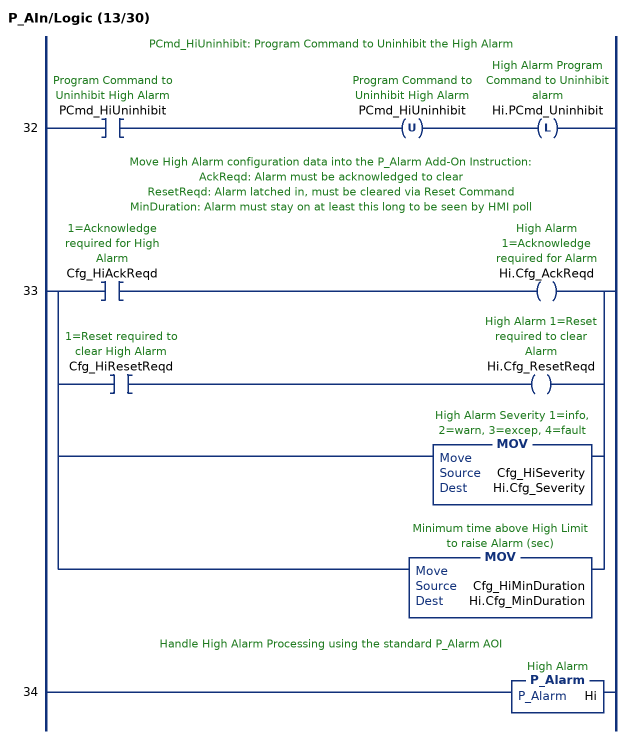
   // PCmd_HiUninhibit: Program Command to Uninhibit the High Alarm
   32: XIC(PCmd_HiUninhibit)OTU(PCmd_HiUninhibit)OTL(Hi.PCmd_Uninhibit);
   // Move High Alarm configuration data into the P_Alarm Add-On Instruction:
   // AckReqd: Alarm must be acknowledged to clear
   // ResetReqd: Alarm latched in, must be cleared via Reset Command
   // MinDuration: Alarm must stay on at least this long to be seen by HMI poll
   33: [XIC(Cfg_HiAckReqd) OTE(Hi.Cfg_AckReqd) ,XIC(Cfg_HiResetReqd) OTE(Hi.Cfg_ResetReqd) ,MOV(Cfg_HiSeverity,Hi.Cfg_Severity) ,MOV(Cfg_HiMinDuration,Hi.Cfg_MinDuration) ];
   // Handle High Alarm Processing using the standard P_Alarm AOI
   34: P_Alarm(Hi);
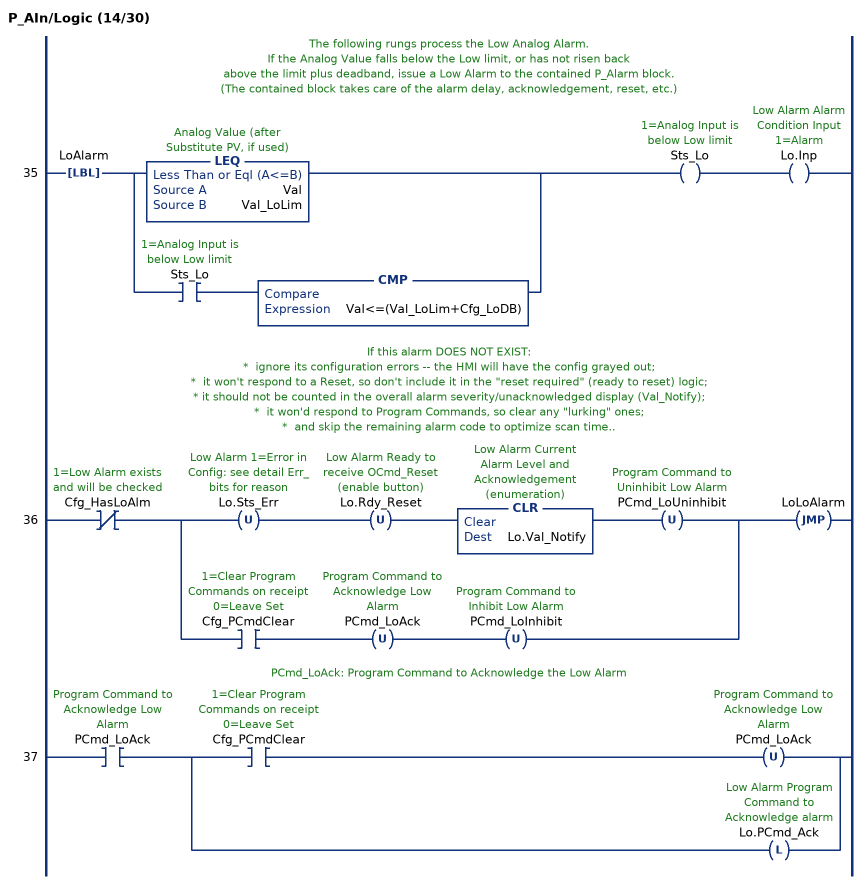
   // The following rungs process the Low Analog Alarm.
   // If the Analog Value falls below the Low limit, or has not risen back
   // above the limit plus deadband, issue a Low Alarm to the contained P_Alarm block.
   // (The contained block takes care of the alarm delay, acknowledgement, reset, etc.)
   35: LBL(LoAlarm)[LEQ(Val,Val_LoLim) ,XIC(Sts_Lo) CMP(Val<=(Val_LoLim+Cfg_LoDB)) ]OTE(Sts_Lo)OTE(Lo.Inp);
   // If this alarm DOES NOT EXIST:
   // *  ignore its configuration errors -- the HMI will have the config grayed out;
   // *  it won't respond to a Reset, so don't include it in the "reset required" (ready to reset) logic;
   // * it should not be counted in the overall alarm severity/unacknowledged display (Val_Notify);
   // *  it won'd respond to Program Commands, so clear any "lurking" ones;
   // *  and skip the remaining alarm code to optimize scan time..
   36: XIO(Cfg_HasLoAlm)[OTU(Lo.Sts_Err) OTU(Lo.Rdy_Reset) CLR(Lo.Val_Notify) OTU(PCmd_LoUninhibit) ,XIC(Cfg_PCmdClear) OTU(PCmd_LoAck) OTU(PCmd_LoInhibit) ]JMP(LoLoAlarm);
   // PCmd_LoAck: Program Command to Acknowledge the Low Alarm
   37: XIC(PCmd_LoAck)[XIC(Cfg_PCmdClear) OTU(PCmd_LoAck) ,OTL(Lo.PCmd_Ack) ];
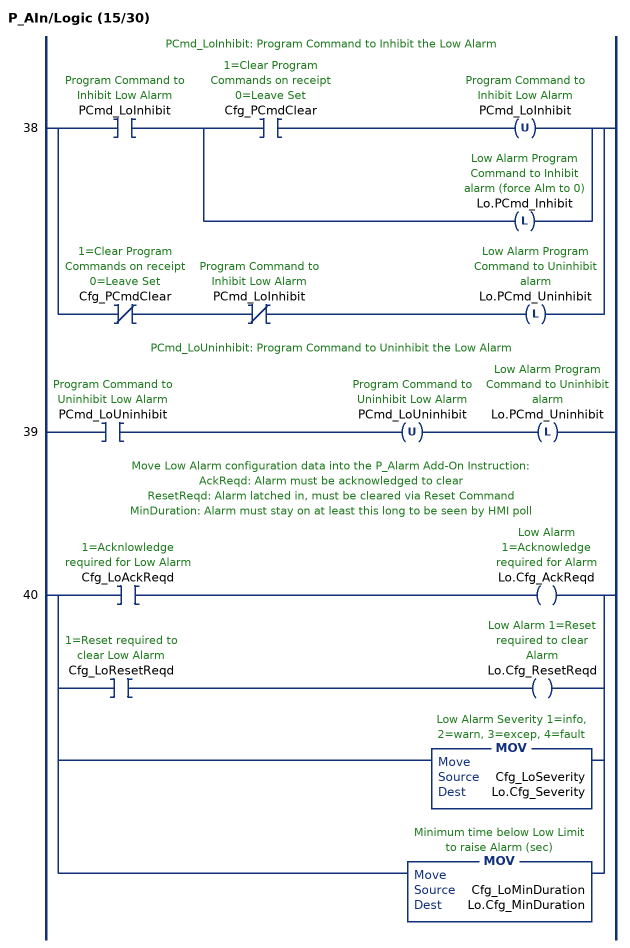
   // PCmd_LoInhibit: Program Command to Inhibit the Low Alarm
   38: [XIC(PCmd_LoInhibit) [XIC(Cfg_PCmdClear) OTU(PCmd_LoInhibit) ,OTL(Lo.PCmd_Inhibit) ] ,XIO(Cfg_PCmdClear) XIO(PCmd_LoInhibit) OTL(Lo.PCmd_Uninhibit) ];
   // PCmd_LoUninhibit: Program Command to Uninhibit the Low Alarm
   39: XIC(PCmd_LoUninhibit)OTU(PCmd_LoUninhibit)OTL(Lo.PCmd_Uninhibit);
   // Move Low Alarm configuration data into the P_Alarm Add-On Instruction:
   // AckReqd: Alarm must be acknowledged to clear
   // ResetReqd: Alarm latched in, must be cleared via Reset Command
   // MinDuration: Alarm must stay on at least this long to be seen by HMI poll
   40: [XIC(Cfg_LoAckReqd) OTE(Lo.Cfg_AckReqd) ,XIC(Cfg_LoResetReqd) OTE(Lo.Cfg_ResetReqd) ,MOV(Cfg_LoSeverity,Lo.Cfg_Severity) ,MOV(Cfg_LoMinDuration,Lo.Cfg_MinDuration) ];
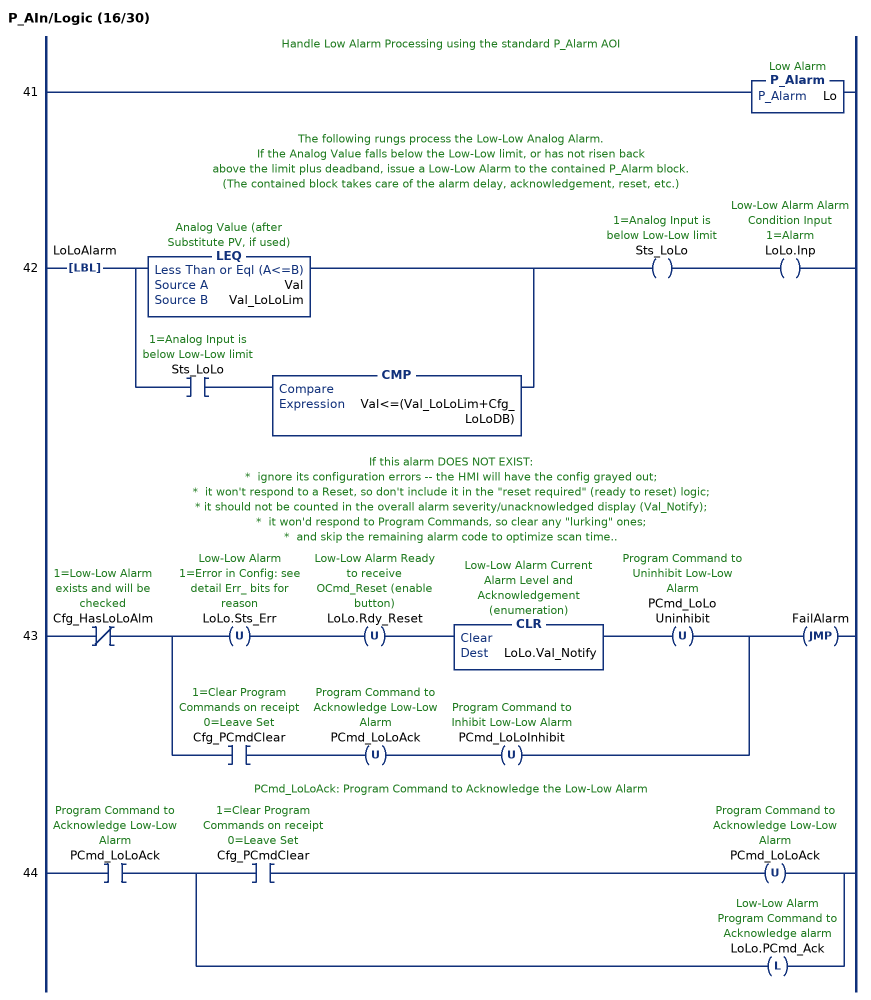
   // Handle Low Alarm Processing using the standard P_Alarm AOI
   41: P_Alarm(Lo);
   // The following rungs process the Low-Low Analog Alarm.
   // If the Analog Value falls below the Low-Low limit, or has not risen back
   // above the limit plus deadband, issue a Low-Low Alarm to the contained P_Alarm block.
   // (The contained block takes care of the alarm delay, acknowledgement, reset, etc.)
   42: LBL(LoLoAlarm)[LEQ(Val,Val_LoLoLim) ,XIC(Sts_LoLo) CMP(Val<=(Val_LoLoLim+Cfg_LoLoDB)) ]OTE(Sts_LoLo)OTE(LoLo.Inp);
   // If this alarm DOES NOT EXIST:
   // *  ignore its configuration errors -- the HMI will have the config grayed out;
   // *  it won't respond to a Reset, so don't include it in the "reset required" (ready to reset) logic;
   // * it should not be counted in the overall alarm severity/unacknowledged display (Val_Notify);
   // *  it won'd respond to Program Commands, so clear any "lurking" ones;
   // *  and skip the remaining alarm code to optimize scan time..
   43: XIO(Cfg_HasLoLoAlm)[OTU(LoLo.Sts_Err) OTU(LoLo.Rdy_Reset) CLR(LoLo.Val_Notify) OTU(PCmd_LoLoUninhibit) ,XIC(Cfg_PCmdClear) OTU(PCmd_LoLoAck) OTU(PCmd_LoLoInhibit) ]JMP(FailAlarm);
   // PCmd_LoLoAck: Program Command to Acknowledge the Low-Low Alarm
   44: XIC(PCmd_LoLoAck)[XIC(Cfg_PCmdClear) OTU(PCmd_LoLoAck) ,OTL(LoLo.PCmd_Ack) ];
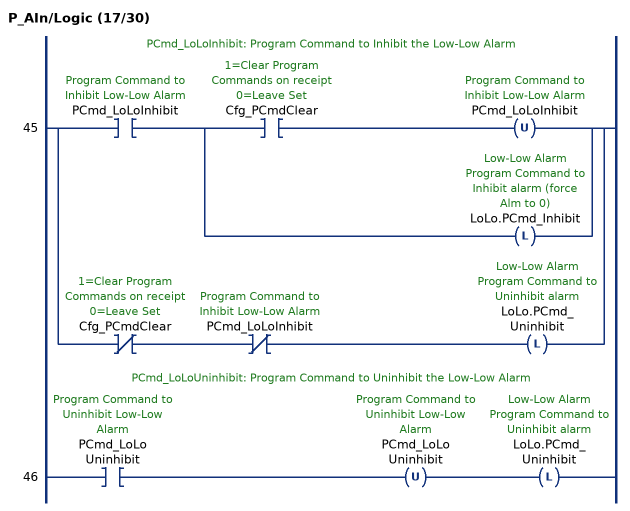
   // PCmd_LoLoInhibit: Program Command to Inhibit the Low-Low Alarm
   45: [XIC(PCmd_LoLoInhibit) [XIC(Cfg_PCmdClear) OTU(PCmd_LoLoInhibit) ,OTL(LoLo.PCmd_Inhibit) ] ,XIO(Cfg_PCmdClear) XIO(PCmd_LoLoInhibit) OTL(LoLo.PCmd_Uninhibit) ];
   // PCmd_LoLoUninhibit: Program Command to Uninhibit the Low-Low Alarm
   46: XIC(PCmd_LoLoUninhibit)OTU(PCmd_LoLoUninhibit)OTL(LoLo.PCmd_Uninhibit);
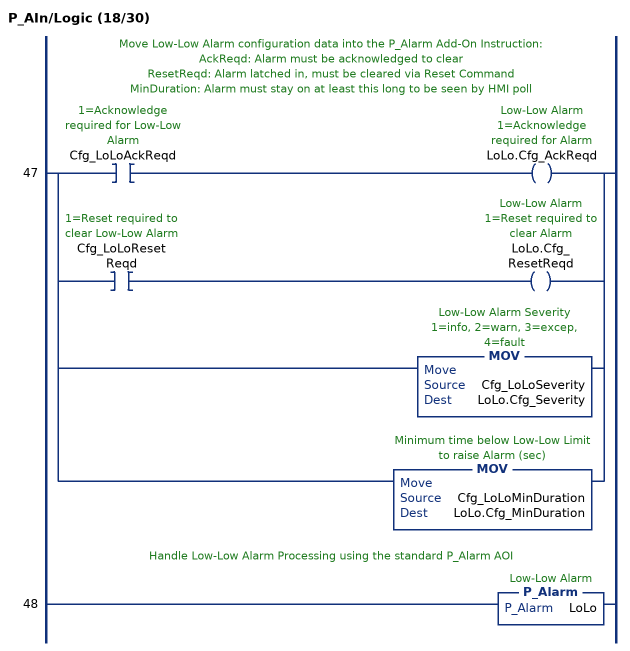
   // Move Low-Low Alarm configuration data into the P_Alarm Add-On Instruction:
   // AckReqd: Alarm must be acknowledged to clear
   // ResetReqd: Alarm latched in, must be cleared via Reset Command
   // MinDuration: Alarm must stay on at least this long to be seen by HMI poll
   47: [XIC(Cfg_LoLoAckReqd) OTE(LoLo.Cfg_AckReqd) ,XIC(Cfg_LoLoResetReqd) OTE(LoLo.Cfg_ResetReqd) ,MOV(Cfg_LoLoSeverity,LoLo.Cfg_Severity) ,MOV(Cfg_LoLoMinDuration,LoLo.Cfg_MinDuration) ];
   // Handle Low-Low Alarm Processing using the standard P_Alarm AOI
   48: P_Alarm(LoLo);
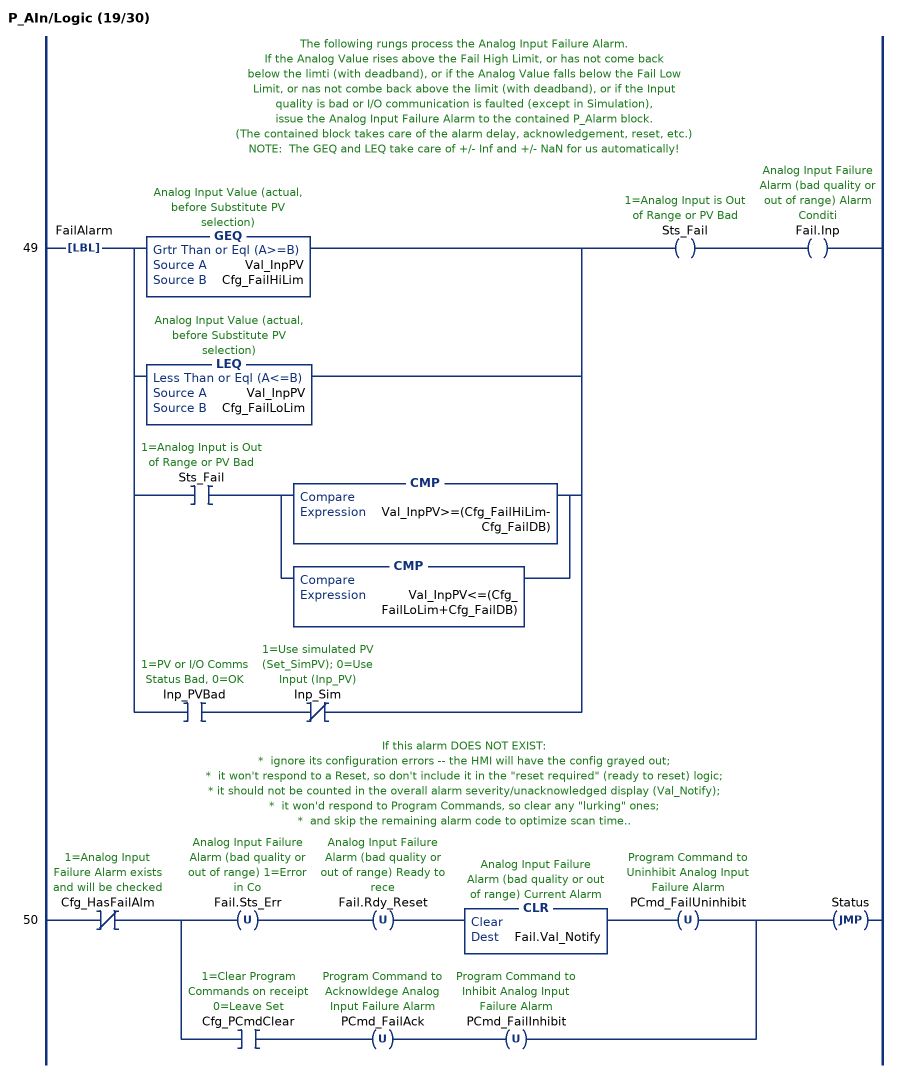
   // The following rungs process the Analog Input Failure Alarm.
   // If the Analog Value rises above the Fail High Limit, or has not come back
   // below the limti (with deadband), or if the Analog Value falls below the Fail Low
   // Limit, or nas not combe back above the limit (with deadband), or if the Input
   // quality is bad or I/O communication is faulted (except in Simulation),
   // issue the Analog Input Failure Alarm to the contained P_Alarm block.
   // (The contained block takes care of the alarm delay, acknowledgement, reset, etc.)
   // NOTE:  The GEQ and LEQ take care of +/- Inf and +/- NaN for us automatically!
   49: LBL(FailAlarm)[GEQ(Val_InpPV,Cfg_FailHiLim) ,LEQ(Val_InpPV,Cfg_FailLoLim) ,XIC(Sts_Fail) [CMP(Val_InpPV>=(Cfg_FailHiLim-Cfg_FailDB)) ,CMP(Val_InpPV<=(Cfg_FailLoLim+Cfg_FailDB)) ] ,XIC(Inp_PVBad) XIO(Inp_Sim) ]OTE(Sts_Fail)OTE(Fail.Inp);
   // If this alarm DOES NOT EXIST:
   // *  ignore its configuration errors -- the HMI will have the config grayed out;
   // *  it won't respond to a Reset, so don't include it in the "reset required" (ready to reset) logic;
   // * it should not be counted in the overall alarm severity/unacknowledged display (Val_Notify);
   // *  it won'd respond to Program Commands, so clear any "lurking" ones;
   // *  and skip the remaining alarm code to optimize scan time..
   50: XIO(Cfg_HasFailAlm)[OTU(Fail.Sts_Err) OTU(Fail.Rdy_Reset) CLR(Fail.Val_Notify) OTU(PCmd_FailUninhibit) ,XIC(Cfg_PCmdClear) OTU(PCmd_FailAck) OTU(PCmd_FailInhibit) ]JMP(Status);
